{attribute addProperty BoxType "EL3483-0060-0018"}
{attribute addProperty Id "VoltageAT %I*REAL324"}
{attribute addProperty CRC "4266836333"}
{attribute addProperty SizeInBites "32"}
{attribute addProperty SizeInBytes "4"}
TYPE L2_Basic_FE52C16D :
STRUCT
	{attribute addProperty Name "Voltage"}
	Voltage AT %I* : REAL;
END_STRUCT
END_TYPE

(* stored: Version 1.2.0.0, ProductVersion 3.1.4024.9
   DUT L2_Basic_FE52C16D: Id {e2b28b1a-9782-4627-be96-3a975adba97a} *)
